FUNCTION_BLOCK FB_Intersection_Test EXTENDS TcUnit.FB_TestSuite
VAR
END_VAR

NewIntersectionStartsInAllRed();
IntersectionAdvancesThroughPhasesInOrder();

METHOD PRIVATE IntersectionAdvancesThroughPhasesInOrder
VAR
	intersection : FB_Intersection;
END_VAR
TEST('IntersectionAdvancesThroughPhasesInOrder');

// starts AllRed
AssertEquals_INT(
    Expected := TO_INT(E_Phase.AllRed),
    Actual   := TO_INT(intersection.CurrentPhase),
    Message  := 'Should start AllRed');

intersection.Advance();           
AssertEquals_INT(
    Expected := TO_INT(E_Phase.NorthSouthFlowing),
    Actual   := TO_INT(intersection.CurrentPhase),
    Message  := 'AllRed should advance to NorthSouthFlowing');

intersection.Advance();
AssertEquals_INT(
    Expected := TO_INT(E_Phase.NorthSouthClearing),
    Actual   := TO_INT(intersection.CurrentPhase),
    Message  := 'NorthSouthFlowing should advance to NorthSouthClearing');

intersection.Advance();
AssertEquals_INT(
    Expected := TO_INT(E_Phase.EastWestFlowing),
    Actual   := TO_INT(intersection.CurrentPhase),
    Message  := 'NorthSouthClearing should advance to EastWestFlowing');

intersection.Advance();
AssertEquals_INT(
    Expected := TO_INT(E_Phase.EastWestClearing),
    Actual   := TO_INT(intersection.CurrentPhase),
    Message  := 'EastWestFlowing should advance to EastWestClearing');

intersection.Advance();
AssertEquals_INT(
    Expected := TO_INT(E_Phase.NorthSouthFlowing),
    Actual   := TO_INT(intersection.CurrentPhase),
    Message  := 'EastWestClearing should wrap to NorthSouthFlowing (not AllRed)');

TEST_FINISHED();
END_METHOD

METHOD PRIVATE NewIntersectionStartsInAllRed
VAR
	intersection : FB_Intersection;
END_VAR
TEST('NewIntersectionStartsInAllRed');

AssertEquals_INT(
    Expected := TO_INT(E_Phase.AllRed),
    Actual   := TO_INT(intersection.CurrentPhase),
    Message  := 'A new intersection should start in AllRed for safety');

TEST_FINISHED();
END_METHOD

END_FUNCTION_BLOCK

(* stored: Version 1.1.0.1, ProductVersion 3.1.4024.12
   POU FB_Intersection_Test: Id {c110743a-9204-448b-b4a8-3ebea3fe05df}, SpecialFunc None
   Method IntersectionAdvancesThroughPhasesInOrder: Id {5843715c-18fa-49a6-a054-df0239c4a384}
   Method NewIntersectionStartsInAllRed: Id {70909ec8-d067-4845-976a-244e0c3b0421} *)
